VAR_GLOBAL
    sPLCName: STRING[34] := 'Crate_000';
    sPLCVersion: STRING[34] := '0.9.3';
    sPLCAuthor1: STRING[34] := 'ESS Lund';
    sPLCAuthor2: STRING[34] := 'ESS Lund';

//PILS Devices
//First available memory area for PILS devices is 104. 64-99 is used by the indexer
//Run the python script "check_fix_gvl_pils.py" to check that the PILS devices have a correct memory allocation

(* Example code to define 2 Axes and other devices:

    stVariable1 AT %MB104: ST_1201;
    stVariable2 AT %MB108: ST_1202;

        //Axis #1 (x stage)
    stMotorM1       AT %MB128: ST_5008;
    fbMotorM1: FB_5008_Axis := (nPILSDeviceNumber := 3);
    stMotorM1Param: ST_AxisParameters;
    stMotorM1ErrorID AT %MB144: ST_1202;
    stMotorM1EncoderRaw AT %MB148: ST_1202;

        //Axis #2

    stMotorM2 AT %MB152: ST_5010;
    fbMotorM2: FB_5010_Axis := (nPILSDeviceNumber := 5);
    stMotorM2Param: ST_AxisParameters;
    stMotor2Temp AT %MB184: ST_1302;
    stMotorM2EncoderRaw AT %MB188: ST_1202;
*)

// Array of Devices
// Modify the array to fit the number of devices you have
// nUnit codes: mm = 16xfd04, degrees = 16x000C, Celsius =16x0009, Kelvin 16x0008

    astDevices: ARRAY [1..8] OF ST_DeviceInfo :=[
        (nTypCode := 16#1201, sName := 'Variable1', nOffset := 104),
        (nTypCode := 16#1202, sName := 'Variable2', nOffset := 108),
        (nTypCode := 16#5008, sName := 'M1 Example', nOffset := 128, nUnit := 16#FD04, asAUX := [('notHomed'),('inTargetPos'),('enabled'),('localMode')], nFlags := 1, sDESC := 'Motor M1'),
        (nTypCode := 16#1202, sName := 'errorID', nOffset := 144),
        (nTypCode := 16#1202, sName := 'encoder1Raw', nOffset := 148),
        (nTypCode := 16#5010, sName := 'M2 Example', nOffset := 152, nUnit := 16#FD04, asAUX := [(''),(''),(''),(''),(''),(''),(''),(''),(''),(''),(''),(''),(''),(''),(''),(''),(''),('InterlockFwd'),('InterlockBwd'),('localMode'),('inTargetPos'),('homeSensor'),('notHomed'),('enabled')], nFlags := 1),
        (nTypCode := 16#1302, sName := 'Temp#2', nOffset := 184, nUnit := 16#0009),
        (nTypCode := 16#1202, sName := 'encoder2Raw', nOffset := 188)];
END_VAR

(* stored: Version 1.1.0.1, ProductVersion 3.1.4024.5
   GVL GVL_PILS: Id {ace53d5e-03a7-4e79-9a33-72de579eb8fd} *)
